PROGRAM Axis03_Auto
VAR
//System_Bit
	Always_ON	:	BOOL	:=TRUE	;//상시 ON 
	Always_OFF	:	BOOL	:=FALSE	;//상시 OFF
END_VAR

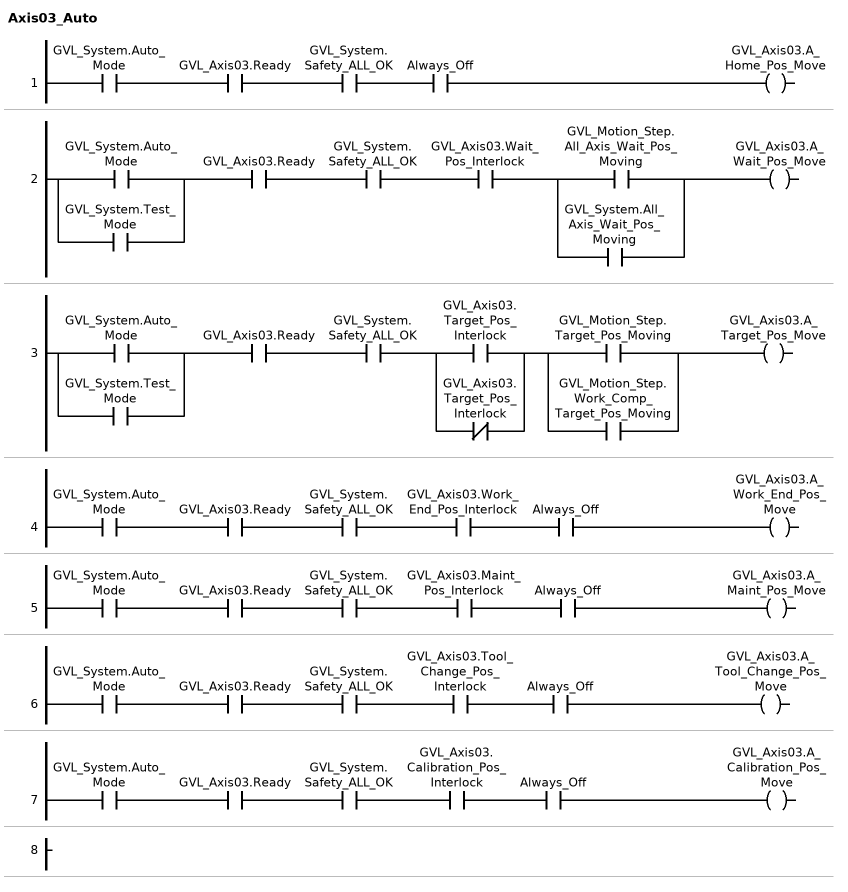
// NETWORK 1
GVL_Axis03.A_Home_Pos_Move := GVL_System.Auto_Mode AND GVL_Axis03.Ready AND GVL_System.Safety_ALL_OK AND Always_Off;

// NETWORK 2
GVL_Axis03.A_Wait_Pos_Move := (GVL_System.Auto_Mode OR GVL_System.Test_Mode) AND GVL_Axis03.Ready AND GVL_System.Safety_ALL_OK AND GVL_Axis03.Wait_Pos_Interlock AND (GVL_Motion_Step.All_Axis_Wait_Pos_Moving OR GVL_System.All_Axis_Wait_Pos_Moving);

// NETWORK 3
GVL_Axis03.A_Target_Pos_Move := (GVL_System.Auto_Mode OR GVL_System.Test_Mode) AND GVL_Axis03.Ready AND GVL_System.Safety_ALL_OK AND (GVL_Axis03.Target_Pos_Interlock OR NOT GVL_Axis03.Target_Pos_Interlock) AND (GVL_Motion_Step.Target_Pos_Moving OR GVL_Motion_Step.Work_Comp_Target_Pos_Moving);

// NETWORK 4
GVL_Axis03.A_Work_End_Pos_Move := GVL_System.Auto_Mode AND GVL_Axis03.Ready AND GVL_System.Safety_ALL_OK AND GVL_Axis03.Work_End_Pos_Interlock AND Always_Off;

// NETWORK 5
GVL_Axis03.A_Maint_Pos_Move := GVL_System.Auto_Mode AND GVL_Axis03.Ready AND GVL_System.Safety_ALL_OK AND GVL_Axis03.Maint_Pos_Interlock AND Always_Off;

// NETWORK 6
GVL_Axis03.A_Tool_Change_Pos_Move := GVL_System.Auto_Mode AND GVL_Axis03.Ready AND GVL_System.Safety_ALL_OK AND GVL_Axis03.Tool_Change_Pos_Interlock AND Always_Off;

// NETWORK 7
GVL_Axis03.A_Calibration_Pos_Move := GVL_System.Auto_Mode AND GVL_Axis03.Ready AND GVL_System.Safety_ALL_OK AND GVL_Axis03.Calibration_Pos_Interlock AND Always_Off;

// NETWORK 8

END_PROGRAM

(* stored: Version 1.1.0.1, ProductVersion 3.1.4024.15
   POU Axis03_Auto: Id {2964529e-7d2c-466b-a161-e686778cebf0}, SpecialFunc None *)
